FUNCTION_BLOCK SENSORS_ACTUATORS (* Composite Function Block Type *)
  (* Standard: 61499-2 *)
  (* Version 1.0, 2019-03-29, adeel *)
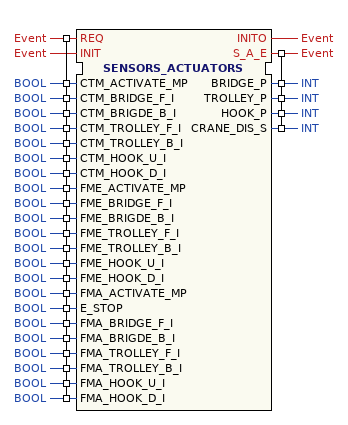
  EVENT_INPUT
    REQ WITH CTM_TROLLEY_F_I, FMA_BRIGDE_B_I, FMA_HOOK_D_I, FMA_TROLLEY_F_I, FMA_HOOK_U_I, FMA_TROLLEY_B_I, FMA_BRIDGE_F_I, CTM_TROLLEY_B_I, FMA_ACTIVATE_MP, CTM_HOOK_U_I, FME_HOOK_D_I, CTM_HOOK_D_I, FME_HOOK_U_I, FME_ACTIVATE_MP, FME_TROLLEY_B_I, FME_BRIDGE_F_I, FME_TROLLEY_F_I, FME_BRIGDE_B_I, CTM_BRIGDE_B_I, CTM_BRIDGE_F_I, CTM_ACTIVATE_MP, E_STOP; (* Normal Execution Request *)
    INIT; (* Initialization Request *)
  END_EVENT
  EVENT_OUTPUT
    INITO; (* Initialization Confirm *)
    S_A_E WITH BRIDGE_P, TROLLEY_P, CRANE_DIS_S, HOOK_P; (* sensors and actuators event *)
  END_EVENT
  VAR_INPUT
    CTM_ACTIVATE_MP : BOOL;
    CTM_BRIDGE_F_I : BOOL;
    CTM_BRIGDE_B_I : BOOL;
    CTM_TROLLEY_F_I : BOOL;
    CTM_TROLLEY_B_I : BOOL;
    CTM_HOOK_U_I : BOOL;
    CTM_HOOK_D_I : BOOL;
    FME_ACTIVATE_MP : BOOL;
    FME_BRIDGE_F_I : BOOL;
    FME_BRIGDE_B_I : BOOL;
    FME_TROLLEY_F_I : BOOL;
    FME_TROLLEY_B_I : BOOL;
    FME_HOOK_U_I : BOOL;
    FME_HOOK_D_I : BOOL;
    FMA_ACTIVATE_MP : BOOL;
    E_STOP : BOOL;
    FMA_BRIDGE_F_I : BOOL;
    FMA_BRIGDE_B_I : BOOL;
    FMA_TROLLEY_F_I : BOOL;
    FMA_TROLLEY_B_I : BOOL;
    FMA_HOOK_U_I : BOOL;
    FMA_HOOK_D_I : BOOL;
  END_VAR
  VAR_OUTPUT
    BRIDGE_P : INT; (* bridge position *)
    TROLLEY_P : INT;
    HOOK_P : INT;
    CRANE_DIS_S : INT; (* crane distance sensor *)
  END_VAR
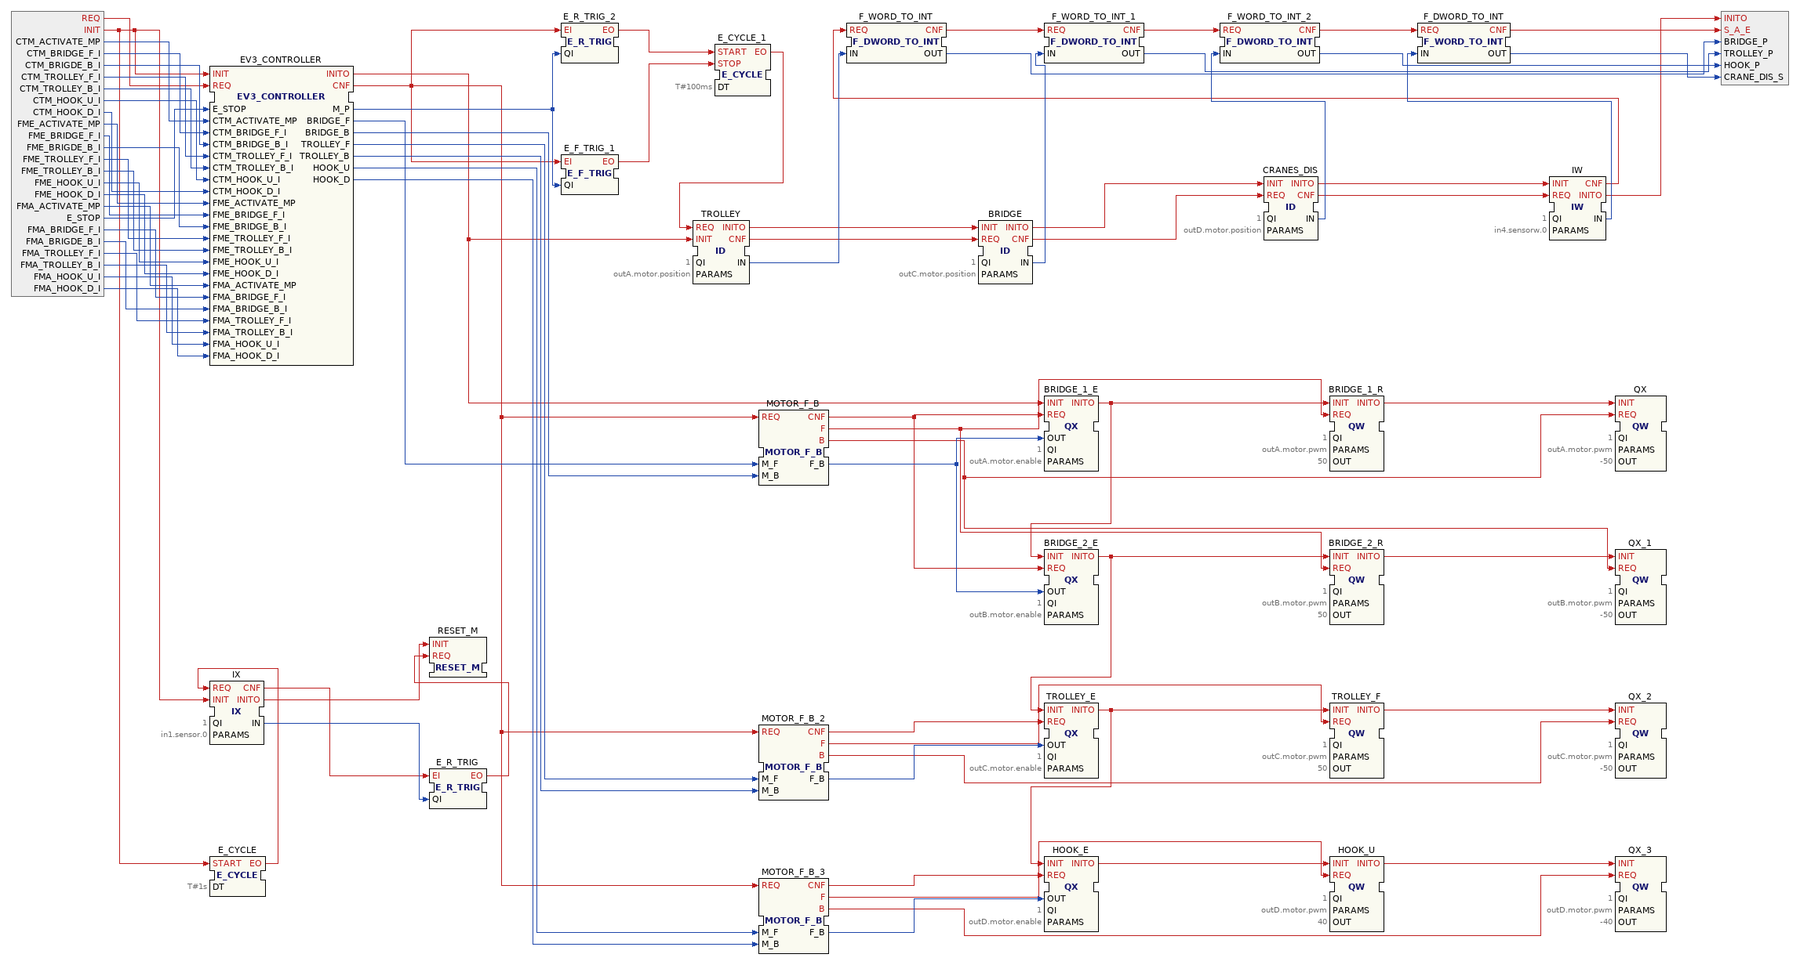
  FBS
    HOOK_U : QW(QI := 1, PARAMS := outD.motor.pwm, OUT := 40);
    TROLLEY_F : QW(QI := 1, PARAMS := outC.motor.pwm, OUT := 50);
    BRIDGE_2_R : QW(QI := 1, PARAMS := outB.motor.pwm, OUT := 50);
    BRIDGE_1_R : QW(QI := 1, PARAMS := outA.motor.pwm, OUT := 50);
    BRIDGE_2_E : QX(QI := 1, PARAMS := outB.motor.enable);
    HOOK_E : QX(QI := 1, PARAMS := outD.motor.enable);
    TROLLEY_E : QX(QI := 1, PARAMS := outC.motor.enable);
    BRIDGE_1_E : QX(QI := 1, PARAMS := outA.motor.enable);
    IX : IX(QI := 1, PARAMS := in1.sensor.0);
    E_R_TRIG : E_R_TRIG;
    E_CYCLE : E_CYCLE(DT := T#1s);
    CRANES_DIS : ID(QI := 1, PARAMS := outD.motor.position);
    BRIDGE : ID(QI := 1, PARAMS := outC.motor.position);
    TROLLEY : ID(QI := 1, PARAMS := outA.motor.position);
    F_WORD_TO_INT : F_DWORD_TO_INT;
    F_WORD_TO_INT_1 : F_DWORD_TO_INT;
    F_WORD_TO_INT_2 : F_DWORD_TO_INT;
    QX : QW(QI := 1, PARAMS := outA.motor.pwm, OUT := -50);
    QX_1 : QW(QI := 1, PARAMS := outB.motor.pwm, OUT := -50);
    QX_2 : QW(QI := 1, PARAMS := outC.motor.pwm, OUT := -50);
    QX_3 : QW(QI := 1, PARAMS := outD.motor.pwm, OUT := -40);
    E_F_TRIG_1 : E_F_TRIG;
    E_R_TRIG_2 : E_R_TRIG;
    E_CYCLE_1 : E_CYCLE(DT := T#100ms);
    EV3_CONTROLLER : EV3_CONTROLLER;
    IW : IW(QI := 1, PARAMS := in4.sensorw.0);
    F_DWORD_TO_INT : F_WORD_TO_INT;
    MOTOR_F_B : MOTOR_F_B;
    MOTOR_F_B_2 : MOTOR_F_B;
    MOTOR_F_B_3 : MOTOR_F_B;
    RESET_M : RESET_M;
  END_FBS
  EVENT_CONNECTIONS
    BRIDGE_1_E.INITO TO BRIDGE_1_R.INIT;
    BRIDGE_1_E.INITO TO BRIDGE_2_E.INIT;
    BRIDGE_2_E.INITO TO BRIDGE_2_R.INIT;
    BRIDGE_2_E.INITO TO TROLLEY_E.INIT;
    TROLLEY_E.INITO TO TROLLEY_F.INIT;
    HOOK_E.INITO TO HOOK_U.INIT;
    IX.CNF TO E_R_TRIG.EI;
    E_CYCLE.EO TO IX.REQ;
    INIT TO IX.INIT;
    BRIDGE.INITO TO CRANES_DIS.INIT;
    BRIDGE.CNF TO CRANES_DIS.REQ;
    TROLLEY.INITO TO BRIDGE.INIT;
    TROLLEY.CNF TO BRIDGE.REQ;
    F_WORD_TO_INT.CNF TO F_WORD_TO_INT_1.REQ;
    F_WORD_TO_INT_1.CNF TO F_WORD_TO_INT_2.REQ;
    E_R_TRIG_2.EO TO E_CYCLE_1.START;
    E_CYCLE_1.EO TO TROLLEY.REQ;
    EV3_CONTROLLER.CNF TO E_R_TRIG_2.EI;
    EV3_CONTROLLER.CNF TO E_F_TRIG_1.EI;
    REQ TO EV3_CONTROLLER.REQ;
    INIT TO EV3_CONTROLLER.INIT;
    EV3_CONTROLLER.INITO TO BRIDGE_1_E.INIT;
    EV3_CONTROLLER.INITO TO TROLLEY.INIT;
    CRANES_DIS.INITO TO IW.INIT;
    CRANES_DIS.CNF TO IW.REQ;
    IW.CNF TO F_WORD_TO_INT.REQ;
    IW.INITO TO INITO;
    F_WORD_TO_INT_2.CNF TO F_DWORD_TO_INT.REQ;
    F_DWORD_TO_INT.CNF TO S_A_E;
    EV3_CONTROLLER.CNF TO MOTOR_F_B.REQ;
    MOTOR_F_B.CNF TO BRIDGE_1_E.REQ;
    TROLLEY_E.INITO TO HOOK_E.INIT;
    HOOK_U.INITO TO QX_3.INIT;
    TROLLEY_F.INITO TO QX_2.INIT;
    BRIDGE_2_R.INITO TO QX_1.INIT;
    BRIDGE_1_R.INITO TO QX.INIT;
    MOTOR_F_B.F TO BRIDGE_1_R.REQ;
    MOTOR_F_B.B TO QX.REQ;
    MOTOR_F_B_2.F TO TROLLEY_F.REQ;
    MOTOR_F_B_2.B TO QX_2.REQ;
    MOTOR_F_B_3.F TO HOOK_U.REQ;
    MOTOR_F_B_3.B TO QX_3.REQ;
    MOTOR_F_B_3.CNF TO HOOK_E.REQ;
    MOTOR_F_B.F TO BRIDGE_2_R.REQ;
    MOTOR_F_B.B TO QX_1.REQ;
    MOTOR_F_B_2.CNF TO TROLLEY_E.REQ;
    MOTOR_F_B.CNF TO BRIDGE_2_E.REQ;
    EV3_CONTROLLER.CNF TO MOTOR_F_B_2.REQ;
    EV3_CONTROLLER.CNF TO MOTOR_F_B_3.REQ;
    IX.INITO TO RESET_M.INIT;
    INIT TO E_CYCLE.START;
    E_F_TRIG_1.EO TO E_CYCLE_1.STOP;
    E_R_TRIG.EO TO RESET_M.REQ;
  END_CONNECTIONS
  DATA_CONNECTIONS
    IX.IN TO E_R_TRIG.QI;
    F_WORD_TO_INT.OUT TO BRIDGE_P;
    F_WORD_TO_INT_1.OUT TO TROLLEY_P;
    TROLLEY.IN TO F_WORD_TO_INT.IN;
    BRIDGE.IN TO F_WORD_TO_INT_1.IN;
    CRANES_DIS.IN TO F_WORD_TO_INT_2.IN;
    CTM_ACTIVATE_MP TO EV3_CONTROLLER.CTM_ACTIVATE_MP;
    E_STOP TO EV3_CONTROLLER.E_STOP;
    CTM_BRIDGE_F_I TO EV3_CONTROLLER.CTM_BRIDGE_F_I;
    CTM_TROLLEY_F_I TO EV3_CONTROLLER.CTM_TROLLEY_F_I;
    CTM_TROLLEY_B_I TO EV3_CONTROLLER.CTM_TROLLEY_B_I;
    CTM_HOOK_U_I TO EV3_CONTROLLER.CTM_HOOK_U_I;
    CTM_HOOK_D_I TO EV3_CONTROLLER.CTM_HOOK_D_I;
    FME_ACTIVATE_MP TO EV3_CONTROLLER.FME_ACTIVATE_MP;
    FME_BRIDGE_F_I TO EV3_CONTROLLER.FME_BRIDGE_F_I;
    FME_TROLLEY_F_I TO EV3_CONTROLLER.FME_TROLLEY_F_I;
    FME_TROLLEY_B_I TO EV3_CONTROLLER.FME_TROLLEY_B_I;
    FME_HOOK_U_I TO EV3_CONTROLLER.FME_HOOK_U_I;
    FME_HOOK_D_I TO EV3_CONTROLLER.FME_HOOK_D_I;
    FMA_ACTIVATE_MP TO EV3_CONTROLLER.FMA_ACTIVATE_MP;
    FMA_BRIDGE_F_I TO EV3_CONTROLLER.FMA_BRIDGE_F_I;
    FMA_TROLLEY_F_I TO EV3_CONTROLLER.FMA_TROLLEY_F_I;
    FMA_TROLLEY_B_I TO EV3_CONTROLLER.FMA_TROLLEY_B_I;
    FMA_HOOK_U_I TO EV3_CONTROLLER.FMA_HOOK_U_I;
    FMA_HOOK_D_I TO EV3_CONTROLLER.FMA_HOOK_D_I;
    EV3_CONTROLLER.M_P TO E_F_TRIG_1.QI;
    EV3_CONTROLLER.M_P TO E_R_TRIG_2.QI;
    IW.IN TO F_DWORD_TO_INT.IN;
    F_DWORD_TO_INT.OUT TO CRANE_DIS_S;
    F_WORD_TO_INT_2.OUT TO HOOK_P;
    CTM_BRIGDE_B_I TO EV3_CONTROLLER.CTM_BRIDGE_B_I;
    FMA_BRIGDE_B_I TO EV3_CONTROLLER.FMA_BRIDGE_B_I;
    FME_BRIGDE_B_I TO EV3_CONTROLLER.FME_BRIDGE_B_I;
    MOTOR_F_B.F_B TO BRIDGE_1_E.OUT;
    MOTOR_F_B_2.F_B TO TROLLEY_E.OUT;
    MOTOR_F_B_3.F_B TO HOOK_E.OUT;
    EV3_CONTROLLER.BRIDGE_F TO MOTOR_F_B.M_F;
    EV3_CONTROLLER.BRIDGE_B TO MOTOR_F_B.M_B;
    EV3_CONTROLLER.TROLLEY_F TO MOTOR_F_B_2.M_F;
    EV3_CONTROLLER.TROLLEY_B TO MOTOR_F_B_2.M_B;
    EV3_CONTROLLER.HOOK_U TO MOTOR_F_B_3.M_F;
    EV3_CONTROLLER.HOOK_D TO MOTOR_F_B_3.M_B;
    MOTOR_F_B.F_B TO BRIDGE_2_E.OUT;
  END_CONNECTIONS
END_FUNCTION_BLOCK
